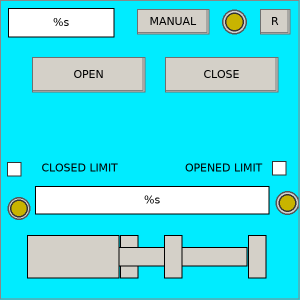
VISUALIZATION vPISTON  // 300x300
VAR_IN_OUT
	PIST1: FB_PISTON;
	
	
END_VAR
    Button (32,57 113x35), "OPEN"
        OnMouseDown: execute { PIST1.bOPEN_CMD:=TRUE; }
    Rectangle (35,186 234x28), "%s", text variable: PIST1.sSTATE
    Lamp1 (6,188 26x41), variable: PIST1.bCLOSED_LIMIT, style: Lamp-Lamp1-Yellow
    Label (30,153 99x30), "CLOSED LIMIT"
    Lamp1 (274,187 27x32), variable: PIST1.bOPEN_LIMIT, style: Lamp-Lamp1-Yellow
    Label (174,153 99x30), "OPENED LIMIT"
    Rectangle (8,8 106x29), "%s", text variable: PIST1.sNAME
    Button (165,57 113x35), "CLOSE"
        OnMouseDown: execute { PIST1.bOPEN_CMD:=FALSE; }
    Button (137,9 72x25), "MANUAL", colour toggle: PIST1.bLOCAL_MANUAL
        toggle PIST1.bLOCAL_MANUAL
    Lamp1 (219,8 31x28), variable: PIST1.bLOCAL_MANUAL, style: Lamp-Lamp1-Yellow
    Checkbox (5,154 34x30), variable: PIST1.bCLOSED_LIMIT
    Checkbox (270,153 34x30), variable: PIST1.bOPEN_LIMIT
    Button (260,9 30x25), "R", colour toggle: PIST1.bLOCAL_MANUAL
        tap PIST1.bLOCAL_RESET
    Rectangle (119,247 128x19), invisible if: NOT PIST1.bOPENED
    Rectangle (248,235 18x43), invisible if: NOT PIST1.bOPENED
    Rectangle (120,235 18x43), invisible if: NOT PIST1.bCLOSED
    Rectangle (78,247 92x19), invisible if: NOT PIST1.bBUSY
    Rectangle (164,235 18x43), invisible if: NOT PIST1.bBUSY
    Rectangle (27,235 92x43), colour toggle: PIST1.bERROR
END_VISUALIZATION

(* stored: Version 1.1.0.1, ProductVersion 3.1.4024.12
   Visu vPISTON: Id {2ca2cd44-1f79-4cce-851b-f97b96892909} *)
